// TIA Portal project "Project1" (V17)

(* hardware
DEVICE "S7-1200 station_1"  S7-1200 Station
   slot 0: "Rack_0"  S7-1200 Rack  Rack  V1.0
   slot 1: "PLC_1"  CPU 1214C DC/DC/DC  6ES7 214-1AG40-0XB0  V4.5
*)

// ===== PLC "PLC_1"  CPU 1214C DC/DC/DC =====

VAR_GLOBAL   // PLC tag table "Default tag table"
   "Tag_1" AT %Q0.0 : Bool;
   "Tag_2" AT %I0.0 : Bool;
   "Tag_3" AT %I0.1 : Bool;
   "Tag_4" AT %Q0.1 : Bool;
   "Tag_5" AT %Q0.2 : Bool;
   "Tag_6" AT %Q0.3 : Bool;
   "Tag_7" AT %Q1.0 : Bool;
   "Tag_8" AT %Q2.0 : Bool;
END_VAR

ORGANIZATION_BLOCK "Main"   // OB1, LAD, ProgramCycle
TITLE = "Main Program Sweep (Cycle)"
{ S7_Optimized_Access := 'TRUE' }
VERSION : 0.1
   VAR_INPUT
      Initial_Call : Bool;   // Initial call of this OB
      Remanence : Bool;   // =True, if remanent data are available
   END_VAR
BEGIN
END_ORGANIZATION_BLOCK